// TIA Portal V19 export
DATA_BLOCK "PAC_320_Data"   // DB14
// stored: MemoryReserve 100
   VAR
      ActualData { S7_SetPoint := 'True'} : "udt_PAC3220";
      MES_MeasuringItem { S7_SetPoint := 'True'} : DInt;
      MES_TotalActiveEnergy { ExternalWritable := 'False'} : LReal;
      MES_60sActiveEnergy : LReal;
      TimeStamp : DTL;
      Aux : Struct
         MinTimer : IEC_TIMER;
         MinutePulse { S7_SetPoint := 'True'} : Bool;
      END_STRUCT;
   END_VAR
BEGIN
END_DATA_BLOCK
